(* LS Electric XG5000 project: 241002_자기유지회로_보조메모리 *)
(* PLC LSPLC *)
(* module base 0 slot 0: 입력 모듈:XGI-D21A (DC 24V 입력, 8점 (전류소스/싱크입력)) *)
(* module base 0 slot 1: 출력 모듈:XGQ-RY1A (릴레이 출력, 8점 (2A용, 단독 COM.)) *)

PROGRAM NewProgram (* task: 스캔 프로그램 *)
VAR
    녹색램프 AT %QX0.1.0 : BOOL;
    보조메모리1 AT %MX0 : BOOL; (* 보조메모리 *)
    보조메모리2 AT %MX1 : BOOL;
    푸시버튼3 AT %IX0.0.0 : BOOL;
    푸시버튼4 AT %IX0.0.1 : BOOL;
    푸시버튼5 AT %IX0.0.4 : BOOL;
    푸시버튼6 AT %IX0.0.5 : BOOL;
END_VAR
VAR
    _p1 : BOOL;
END_VAR

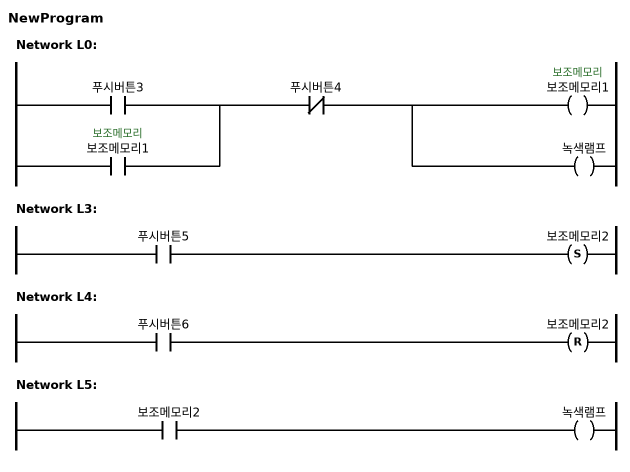
(* Rung L0 *)
_p1 := (푸시버튼3 OR 보조메모리1) AND NOT 푸시버튼4;
보조메모리1 := _p1;
녹색램프 := _p1;
(* Rung L3 *)
IF 푸시버튼5 THEN 보조메모리2 := TRUE; END_IF;
(* Rung L4 *)
IF 푸시버튼6 THEN 보조메모리2 := FALSE; END_IF;
(* Rung L5 *)
녹색램프 := 보조메모리2;
END_PROGRAM